FUNCTION_BLOCK A_Receiver IMPLEMENTS Debug.I_Debug;

//FB_Init is always available implicitly and it is used primarily for initialization.
//The return value is not evaluated. For a specific influence, you can also declare the
//methods explicitly and provide additional code there with the standard initialization
//code. You can evaluate the return value.
METHOD FB_Init: BOOL
VAR_INPUT
    bInitRetains: BOOL; // TRUE: the retain variables are initialized (reset warm / reset cold)
    bInCopyCode: BOOL;  // TRUE: the instance will be copied to the copy code afterward (online change)
	iReceiverList			: I_MutReceiverList;
	iReceiver				: I_Receiver;
END_VAR
IF iReceiverList = 0 THEN
	Debug.DebugMsg(THIS^, ': iReceiverList: Itf = 0!');
	RETURN;
END_IF
IF iReceiver = 0 THEN
	Debug.DebugMsg(THIS^, ': iReceiver: Itf = 0!');
	RETURN;
END_IF

CASE iReceiverList.Push(iReceiver) OF
	Results.Ok:
		// No Error
	Results.None:
		Debug.DebugMsg(iReceiverList, Tc2_Standard.CONCAT(__POUNAME(), ': Tried to insert a double!'));
		Debug.DebugMsg(iReceiver, 'Im a double!');
	Results.Err.Ovf:
		Debug.DebugMsg(iReceiverList, Tc2_Standard.CONCAT(__POUNAME(), ': Overflow!'));
		Debug.DebugMsg(iReceiver, 'Cause of overflow!');
	Results.Err.NoMatch:
		Debug.DebugMsg(iReceiverList, Tc2_Standard.CONCAT(__POUNAME(), ': No Match!'));
		Debug.DebugMsg(iReceiver, 'This already have an owner!');
	ELSE
		Debug.DebugMsg(iReceiverList, Tc2_Standard.CONCAT(__POUNAME(), ': Unknown Error!'));
		Debug.DebugMsg(iReceiver, 'Cause!');		
END_CASE
END_METHOD

METHOD ToDebug : Debug.I_Debug
VAR_INPUT
END_VAR
ToDebug := THIS^;
END_METHOD

END_FUNCTION_BLOCK

(* stored: Version 1.1.0.1
   POU A_Receiver: Id {d221926f-af70-4909-b8df-700990de5bc7}, SpecialFunc None
   Method FB_init: Id {5348752a-bc3e-427a-95de-042541e2ee3d}
   Method ToDebug: Id {4f720a55-07ea-4e24-9d19-4c6b74b6a84f} *)
